Fanuc TP program (LS listing): _TEST_DOOR.LS

/PROG  _TEST_DOOR
/ATTR
OWNER		= MNEDITOR;
COMMENT		= "";
PROG_SIZE	= 285;
CREATE		= DATE 16-10-18  TIME 00:24:46;
MODIFIED	= DATE 16-10-18  TIME 00:26:58;
FILE_NAME	= TEST_DOO;
VERSION		= 0;
LINE_COUNT	= 5;
MEMORY_SIZE	= 785;
PROTECT		= READ_WRITE;
TCD:  STACK_SIZE	= 0,
      TASK_PRIORITY	= 50,
      TIME_SLICE	= 0,
      BUSY_LAMP_OFF	= 0,
      ABORT_REQUEST	= 0,
      PAUSE_REQUEST	= 0;
DEFAULT_GROUP	= *,1,*,*,*;
CONTROL_CODE	= 00000000 00000000;
/APPL
/APPL

AUTO_SINGULARITY_HEADER;
  ENABLE_SINGULARITY_AVOIDANCE   : TRUE;
/MN
   1:  LBL[1] ;
   2:  CALL _OPEN_DOOR    ;
   3:  WAIT   1.00(sec) ;
   4:  CALL _CLOSE_DOOR    ;
   5:  JMP LBL[1] ;
/POS
/END
